FUNCTION_BLOCK CROSSCOMM_PEER_246902A2E9B15C94D (* Service Interface Function Block Type *)
  (* Standard: 61499-2 *)
  (* Version 0.0, 9/22/2017, bababen, nxtControl GmbH, template *)
  PACKAGE Main;
  (* Compiler Cpp nxtControl builtin 1.0 *)
  {SET_ATTRIBUTE(Runtime.FBType.ImplementingType, Runtime.System#DYNGEN_CROSSCOMM_PEER)}
  {SET_ATTRIBUTE(Configuration.GenericFBType.InterfaceParams, Runtime.System#<InterfaceList> <EventOutputs> <Event Name="INITO" /> <Event Name="CNF"> <With Var="RetractLift" /> <With Var="ExtendLift" /> </Event> </EventOutputs> <OutputVars> <VarDeclaration Name="RetractLift" Type="BOOL" /> <VarDeclaration Name="ExtendLift" Type="BOOL" /> </OutputVars> </InterfaceList>)}
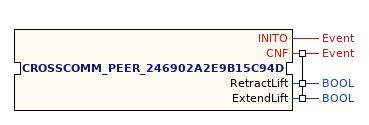
  EVENT_OUTPUT
    INITO;
    CNF WITH RetractLift, ExtendLift;
  END_EVENT
  VAR_OUTPUT
    RetractLift : BOOL;
    ExtendLift : BOOL;
  END_VAR
  EC_STATES
    START;
  END_STATES
END_FUNCTION_BLOCK
